{attribute addProperty BoxType "EJ5101-0000-0016"}
{attribute addProperty Id "Enable_latch_CBIT10.1251Enable_latch_extern_on_positive_edgeBIT10.1252Set_counterBIT10.1253Enable_latch_extern_on_negative_edgeBIT10.1254"}
{attribute addProperty CRC "951080136"}
{attribute addProperty SizeInBites "16"}
{attribute addProperty SizeInBytes "2"}
TYPE Control_38B054C8 :
STRUCT
	{attribute addProperty Name "Enable_latch_C"}
	Enable_latch_C : BOOL;
	{attribute addProperty Name "Enable_latch_extern_on_positive_edge"}
	Enable_latch_extern_on_positive_edge : BOOL;
	{attribute addProperty Name "Set_counter"}
	Set_counter : BOOL;
	{attribute addProperty Name "Enable_latch_extern_on_negative_edge"}
	Enable_latch_extern_on_negative_edge : BOOL;
	{attribute 'hide'}
	reserve_1_BIT_0 : BOOL;
	{attribute 'hide'}
	reserve_1_BIT_1 : BOOL;
	{attribute 'hide'}
	reserve_1_BIT_2 : BOOL;
	{attribute 'hide'}
	reserve_1_BIT_3 : BOOL;
	{attribute 'hide'}
	reserve_2 : BYTE;
END_STRUCT
END_TYPE

(* stored: Version 1.2.0.0, ProductVersion 3.1.4024.9
   DUT Control_38B054C8: Id {f26f52bc-b6b2-4d4e-be2c-37fde7d47422} *)
